ABB RobotStudio station: pathSolution.rsstn

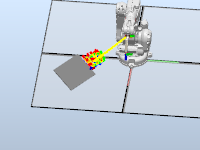
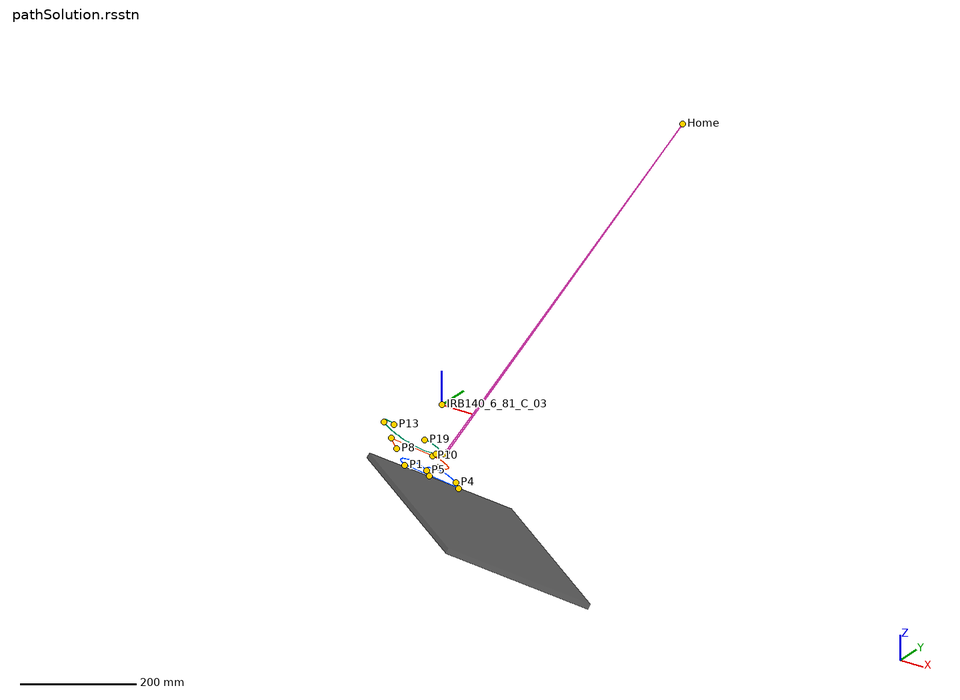
[picture v1: parts stored in the station drawn from their meshes, with robot base, taught points and paths (robot models come from the ABB library and are not in the file)]
Station pathSolution (saved by RobotStudio 22.1.9826.0)
Controller IRB140_6_81
  mechanical unit ROB_1: IRB140_6_81_C_03, 6 joints, base frame (0, 0, 0) mm
Layout (positions relative to the parent item):
  - IRB140_6_81_C_03 [mechanism, from Robots\IRB140_6_81_C_G_03.rslib] at (0, 0, 0) mm; joint values [0, 0, 0, -3.1416, -0.5236, 3.1416] (rad or m)
  - markerTool [mechanism, from Libraries\markerTool.rslib] at (506.29, 0, 679.5) mm, rotated rx 180 ry 60 rz 180 deg
  - Part_1 [part] at (724.73, -597.47, 50) mm, rotated rx 0 ry 0 rz 144.91 deg, size 400 x 264.8 x 158.7 mm
Attachment: markerTool is attached to IRB140_6_81_C_03 / Link6
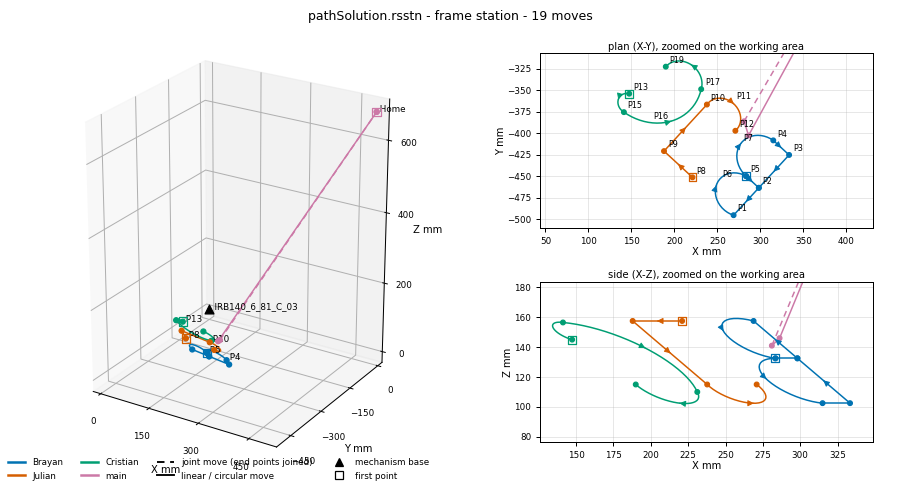
[picture p0: tool path of pathSolution.rsstn in frame station, 19 of 19 moves have a stored position in this frame; points joined in program order, loops and branches not executed]
Targets, tools, work objects and paths stored in the station, written as RAPID:
! task T_ROB1
MODULE CalibData
  PERS tooldata TipBJC:=[TRUE,[[12.254,-0.002,214.736],[0.923879533,0,0.382683432,0]],[0.162,[-27.13,0,109.8621],[1,0,0,0],0.003,0.003,0.0003162]];
  TASK PERS wobjdata whiteBoard:=[FALSE,TRUE,"",[[373.72422246,-432.807039289,90.000000038],[0.351258535,0.094119441,0.24109921,0.899794501]],[[0,0,0],[1,0,0,0]]];
ENDMODULE

! task T_ROB1
MODULE Module1
  CONST robtarget P1:=[[35,135,0],[0,0.707106781,0.707106781,0],[0,-1,0,1],[9E+09,9E+09,9E+09,9E+09,9E+09,9E+09]];
  CONST robtarget P2:=[[35,85,0],[0,0.707106781,0.707106781,0],[0,-1,0,1],[9E+09,9E+09,9E+09,9E+09,9E+09,9E+09]];
  CONST robtarget P3:=[[35,25,0],[0,0.707106781,0.707106781,0],[0,-1,0,1],[9E+09,9E+09,9E+09,9E+09,9E+09,9E+09]];
  CONST robtarget P4:=[[60,25,0],[0,0.707106781,0.707106781,0],[0,-1,0,1],[9E+09,9E+09,9E+09,9E+09,9E+09,9E+09]];
  CONST robtarget P5:=[[55,85,0],[0,0.707106781,0.707106781,0],[0,-1,0,1],[9E+09,9E+09,9E+09,9E+09,9E+09,9E+09]];
  CONST robtarget P6:=[[75,115,0],[0,0.707106781,0.707106781,0],[0,-1,0,1],[9E+09,9E+09,9E+09,9E+09,9E+09,9E+09]];
  CONST robtarget P7:=[[85,60,0],[0,0.707106781,0.707106781,0],[0,-1,0,1],[9E+09,9E+09,9E+09,9E+09,9E+09,9E+09]];
  CONST robtarget Home:=[[506.292,0,679.5],[0.5,0,0.866025404,0],[0,-1,0,1],[9E+09,9E+09,9E+09,9E+09,9E+09,9E+09]];
  CONST robtarget P8:=[[100,135,0],[0,0.707106781,0.707106781,0],[0,-1,0,1],[9E+09,9E+09,9E+09,9E+09,9E+09,9E+09]];
  CONST robtarget P9:=[[145,135,0],[0,0.707106781,0.707106781,0],[0,-1,0,1],[9E+09,9E+09,9E+09,9E+09,9E+09,9E+09]];
  CONST robtarget P10:=[[145,50,0],[0,0.707106781,0.707106781,0],[0,-1,0,1],[9E+09,9E+09,9E+09,9E+09,9E+09,9E+09]];
  CONST robtarget P11:=[[125,25,0],[0,0.707106781,0.707106781,0],[0,-1,0,1],[9E+09,9E+09,9E+09,9E+09,9E+09,9E+09]];
  CONST robtarget P12:=[[100,50,0],[0,0.707106781,0.707106781,0],[0,-1,0,1],[9E+09,9E+09,9E+09,9E+09,9E+09,9E+09]];
  CONST robtarget P7u:=[[85,60,30],[0,0.707106781,0.707106781,0],[0,-1,0,1],[9E+09,9E+09,9E+09,9E+09,9E+09,9E+09]];
  CONST robtarget P17:=[[162,40,0],[0,0.707106781,0.707106781,0],[0,-1,0,1],[9E+09,9E+09,9E+09,9E+09,9E+09,9E+09]];
  CONST robtarget P19:=[[210,50,0],[0,0.707106781,0.707106781,0],[0,-1,0,1],[9E+09,9E+09,9E+09,9E+09,9E+09,9E+09]];
  CONST robtarget P15:=[[210,133,0],[0,0.707106781,0.707106781,0],[0,-1,0,1],[9E+09,9E+09,9E+09,9E+09,9E+09,9E+09]];
  CONST robtarget P14:=[[225,125,0],[0,0.707106781,0.707106781,0],[0,-1,0,1],[9E+09,9E+09,9E+09,9E+09,9E+09,9E+09]];
  CONST robtarget P13:=[[220,110,0],[0,0.707106781,0.707106781,0],[0,-1,0,1],[9E+09,9E+09,9E+09,9E+09,9E+09,9E+09]];
  CONST robtarget P18:=[[190,25,0],[0,0.707106781,0.707106781,0],[0,-1,0,1],[9E+09,9E+09,9E+09,9E+09,9E+09,9E+09]];
  CONST robtarget P16:=[[180,120,0],[0,0.707106781,0.707106781,0],[0,-1,0,1],[9E+09,9E+09,9E+09,9E+09,9E+09,9E+09]];
  CONST robtarget P12u:=[[100,50,30],[0,0.707106781,0.707106781,0],[0,-1,0,1],[9E+09,9E+09,9E+09,9E+09,9E+09,9E+09]];
  PROC Brayan()
    MoveJ P5,v1000,z0,TipBJC\WObj:=whiteBoard;
    MoveL P2,v100,z0,TipBJC\WObj:=whiteBoard;
    MoveL P1,v100,z0,TipBJC\WObj:=whiteBoard;
    MoveC P6,P5,v100,z0,TipBJC\WObj:=whiteBoard;
    MoveC P7,P4,v100,z0,TipBJC\WObj:=whiteBoard;
    MoveL P3,v100,z0,TipBJC\WObj:=whiteBoard;
    MoveL P2,v100,z0,TipBJC\WObj:=whiteBoard;
  ENDPROC
  PROC Julian()
    MoveJ P8,v1000,z0,TipBJC\WObj:=whiteBoard;
    MoveL P9,v100,z0,TipBJC\WObj:=whiteBoard;
    MoveL P10,v100,z0,TipBJC\WObj:=whiteBoard;
    MoveC P11,P12,v100,z0,TipBJC\WObj:=whiteBoard;
  ENDPROC
  PROC Cristian()
    MoveJ P13,v1000,z0,TipBJC\WObj:=whiteBoard;
    MoveC P14,P15,v100,z0,TipBJC\WObj:=whiteBoard;
    MoveC P16,P17,v100,z0,TipBJC\WObj:=whiteBoard;
    MoveC P18,P19,v100,z0,TipBJC\WObj:=whiteBoard;
  ENDPROC
  PROC main()
    MoveJ Home,v1000,z100,tool0;
    Brayan;
    MoveL P7u,v1000,z0,TipBJC\WObj:=whiteBoard;
    Julian;
    MoveL P12u,v1000,z0,TipBJC\WObj:=whiteBoard;
    Cristian;
    MoveJ Home,v1000,z0,tool0;
  ENDPROC
ENDMODULE

